// TIA Portal V18 program export: 2 tag tables, 0 data types, 2 data blocks, 2 code blocks (in call order from the OBs), 1 instance data blocks

VAR_GLOBAL   // PLC tag table "Default tag table"
   outtt AT %M0.0 : Bool;
END_VAR

VAR_GLOBAL   // PLC tag table "Tag table_1"
   nnn1 AT %MD10 : DInt;
   nnn2 AT %MD14 : DInt;
   nnn3 AT %MD18 : DInt;
   nnn4 AT %MD22 : DInt;
   nnn5 AT %MD26 : DInt;
   nnn6 AT %MD30 : DInt;
   nnn7 AT %MD34 : DInt;
   nnn8 AT %MD38 : DInt;
   nnn9 AT %MD42 : DInt;
END_VAR

DATA_BLOCK "Data_block_1"   // DB1
{ S7_Optimized_Access := 'TRUE' }
VERSION : 0.1
// stored: AutoNumber true, IsOnlyStoredInLoadMemory false, IsRetainMemResEnabled false, IsWriteProtectedInAS false, MemoryReserve 100
   VAR
      tag_1 : Real;
      tag_2 : Real;
      tag_3 : Real;
      tag_4 : Real;
      tag_5 : Real;
      tag_6 : Real;
      tag_7 : Real;
      tag_8 : Real;
      tag_9 : Real;
      tag_10 : Real;
      tag_11 : Real;
      tag_12 : Real;
      tag_13 : Real;
   END_VAR
BEGIN
END_DATA_BLOCK

DATA_BLOCK "Data_block_2"   // DB3
{ S7_Optimized_Access := 'TRUE' }
VERSION : 0.1
// stored: AutoNumber true, IsOnlyStoredInLoadMemory false, IsRetainMemResEnabled false, IsWriteProtectedInAS false, MemoryReserve 100
   VAR
      ar : Array[0..1000] of Time_Of_Day;
   END_VAR
BEGIN
END_DATA_BLOCK

ORGANIZATION_BLOCK "Main"   // OB1, LAD, ProgramCycle
TITLE = "Main Program Sweep (Cycle)"
{ S7_Optimized_Access := 'TRUE' }
VERSION : 0.1
// stored: AutoNumber true, IsIECCheckEnabled false, SetENOAutomatically false
   VAR_INPUT
      Initial_Call : Bool;   // Initial call of this OB
      Remanence : Bool;   // =True, if remanent data are available
   END_VAR
   VAR_TEMP
      qqq : Bool;
      qqqqq : Bool;
   END_VAR
BEGIN

REGION Network 1
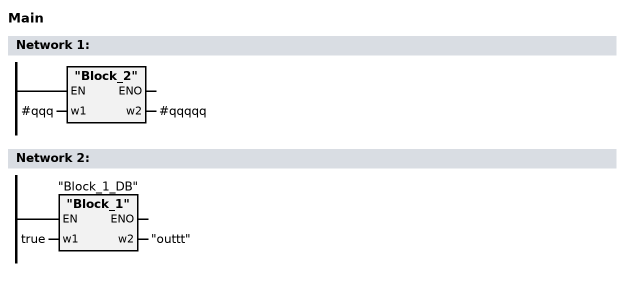
   RUNG wire#powerrail
      "Block_2"(w1 := #qqq, w2 => #qqqqq)
   END_RUNG
   // the same network as SCL:
   "Block_2"(w1 := #qqq, w2 => #qqqqq);
END_REGION

REGION Network 2
   RUNG wire#powerrail
      "Block_1_DB"(w1 := true, w2 => "outtt")
   END_RUNG
   // the same network as SCL:
   "Block_1_DB"(w1 := true, w2 => "outtt");   // "Block_1"
END_REGION
END_ORGANIZATION_BLOCK

FUNCTION "Block_2" : Void   // FC1, LAD
{ S7_Optimized_Access := 'TRUE' }
VERSION : 0.1
// stored: AutoNumber true, IsIECCheckEnabled false, SetENOAutomatically false, UDAEnableTagReadback false
   VAR_INPUT
      w1 : Bool;
   END_VAR
   VAR_OUTPUT
      w2 : Bool;
   END_VAR
BEGIN
END_FUNCTION

DATA_BLOCK "Block_1_DB"   // DB2
VERSION : 0.1
// stored: AutoNumber true, InstanceOfName Block_1, InstanceOfType FB
"Block_1"
   // VAR_INPUT
   //    w1 : Bool;
   // END_VAR
   // VAR_OUTPUT
   //    w2 : Bool;
   // END_VAR
   // VAR
   //    IEC_Timer_0_Instance { S7_SetPoint := 'True'} : TON_TIME;
   // END_VAR
BEGIN
END_DATA_BLOCK
